PROGRAM ReadCSVSecondPractice
VAR
	
	iStep		:eCSVFileReadStep;
	nRow			:INT:=0;
	nColumn			:INT:=0;
	bRead			:BOOL;
	handleFile		:UINT;
	fbFileClose: FB_FileClose;
	fbFileGets: FB_FileGets;
	fbFileOpen: FB_FileOpen;
	fbRead: FB_CSVMemBufferReader;
	FilePath		:STRING:= 'C:\Temp\TextModeGen.csv';
	sCSVLine			:T_MaxString;
	bReadError: BOOL;
	sCSVField: T_MaxString;
END_VAR

CASE iStep OF
	eCSVFileReadStep.iStep_Init:
		IF	bRead THEN 
			bRead := FALSE;
			nRow := 0;
			nColumn := 0;
			MEMSET(ADR(GVL_General.dataArray),0,SIZEOF(GVL_General.dataArray));
			iStep := eCSVFileReadStep.iStep_Open;
		END_IF
		
	eCSVFileReadStep.iStep_Open:	(*prepare to open source file*)
		fbFileOpen(bExecute:=FALSE);
					
		fbFileOpen(sNetId:= ,sPathName:=FilePath ,nMode:= FOPEN_MODEREAD OR FOPEN_MODETEXT,ePath:=PATH_GENERIC ,bExecute:=TRUE,
					tTimeout:=T#3S ,bBusy=> ,bError=> ,nErrId=> ,hFile=> handleFile);
					
		iStep := eCSVFileReadStep.iStep_OpenWait;
		
	eCSVFileReadStep.iStep_OpenWait:

			fbFileOpen(sNetId:= ,sPathName:=FilePath ,nMode:= FOPEN_MODEREAD,ePath:=PATH_GENERIC ,bExecute:=FALSE,
					tTimeout:=T#3S ,bBusy=> ,bError=> ,nErrId=> ,hFile=> handleFile);	
		IF NOT fbFileOpen.bBusy THEN 
			IF NOT fbFileOpen.bError THEN 
				iStep := eCSVFileReadStep.iStep_ReadSingleLine;	
			ELSE
				iStep := eCSVFileReadStep.iStep_CloseOrError;
			END_IF
		END_IF
		
		
	eCSVFileReadStep.iStep_ReadSingleLine:
	
		fbFileGets(sNetId:= ,hFile:=handleFile,bExecute:=FALSE,tTimeout:=T#3S,
					bBusy=> ,bError=> ,nErrId=> ,sLine=> sCSVLine,bEOF=> );
					
		fbFileGets(sNetId:= ,hFile:=handleFile,bExecute:=TRUE,tTimeout:=T#3S,
					bBusy=> ,bError=> ,nErrId=> ,sLine=>sCSVLine,bEOF=> );
					
		fbFileGets(sNetId:= ,hFile:=handleFile,bExecute:=FALSE,tTimeout:=T#3S,
					bBusy=> ,bError=> ,nErrId=> ,sLine=> sCSVLine,bEOF=> );	
					
		IF NOT fbFileGets.bBusy THEN 
			IF NOT fbFileGets.bError THEN 
				IF fbFileGets.bEOF THEN 
					iStep := eCSVFileReadStep.iStep_CloseOrError;
				END_IF
				//add CRLF to the end of the CSVField
				IF(RIGHT(sCSVLine,1) = '$N') THEN 
					sCSVLine := REPLACE(sCSVLine,'$R$N',2,Len(sCSVLine));
					iStep := eCSVFileReadStep.iStep_ParseSingleLine;
				END_IF				
			ELSE
				iStep := eCSVFileReadStep.iStep_CloseOrError;
			END_IF
		END_IF
		
	eCSVFileReadStep.iStep_ParseSingleLine:
		fbRead.eCmd := eEnumCmd_First;
		REPEAT
			fbRead(pBuffer:=ADR(sCSVLine),cbBuffer:=SIZEOF(sCSVLine),bOk=> , 
				getValue=>sCSVField ,pValue=> ,cbValue=>,bCRLF=> ,cbRead=> );			
			IF	fbRead.bOk THEN 
				fbRead.eCmd := eEnumCmd_Next;
				IF NOT fbRead.bCRLF THEN 
					GVL_General.dataArray[nRow,nColumn] := CSVFIELD_TO_STRING(in:= sCSVField,bQM:= FALSE);
					nColumn :=nColumn + 1;
				ELSE
					nColumn := 0;
					nRow := nRow + 1;
					iStep := eCSVFileReadStep.iStep_ReadSingleLine;
				END_IF
			END_IF
		UNTIL NOT fbRead.bOk
		END_REPEAT		
		
		
	eCSVFileReadStep.iStep_CloseOrError:
		fbFileClose(sNetId:= ,hFile:=handleFile ,bExecute:=FALSE,tTimeout:= ,bBusy=> ,bError=> ,nErrId=> );
		fbFileClose(sNetId:= ,hFile:=handleFile ,bExecute:=TRUE,tTimeout:= ,bBusy=> ,bError=> ,nErrId=> );
		IF NOT fbFileClose.bBusy THEN 
			IF NOT fbFileClose.bError THEN 

				iStep := eCSVFileReadStep.iStep_Init;
			ELSE
				bReadError := TRUE;
			END_IF
		END_IF	
END_CASE

END_PROGRAM

(* stored: Version 1.1.0.1, ProductVersion 3.1.4022.16
   POU ReadCSVSecondPractice: Id {4f6e845f-7504-4b65-a464-f337e80da650}, SpecialFunc None *)
